// TIA Portal V20 export
TYPE "ConvHMICMD"
   STRUCT
      StationOnly : Bool;   // Run Within Station Only
      SafetyTest : Bool;   // Safety Test
      Spare1 : Bool;   // Spare
      Spare2 : Bool;   // Spare
      Spare3 : Bool;   // Spare
      Spare4 : Bool;   // Spare
      Spare5 : Bool;   // Spare
      Spare6 : Bool;   // Spare
      Spare7 : Bool;   // Spare
      Spare8 : Bool;   // Spare
      Spare9 : Bool;   // Spare
      Spare10 : Bool;   // Spare
      Spare11 : Bool;   // Spare
      Spare12 : Bool;   // Spare
      Spare13 : Bool;   // Spare
      Spare14 : Bool;   // Spare
      Spare15 : Bool;   // Spare
      Spare16 : Bool;   // Spare
      Spare17 : Bool;   // Spare
      Spare18 : Bool;   // Spare
      Spare19 : Bool;   // Spare
      Spare20 : Bool;   // Spare
      Spare21 : Bool;   // Spare
      Spare22 : Bool;   // Spare
      Spare23 : Bool;   // Spare
      Spare24 : Bool;   // Spare
      Spare25 : Bool;   // Spare
      Spare26 : Bool;   // Spare
      Spare27 : Bool;   // Spare
      Spare28 : Bool;   // Spare
      Spare29 : Bool;   // Spare
      Spare30 : Bool;   // Spare
   END_STRUCT;
END_TYPE
